REGION Network 7: Step 0 (Idle) - Warned Repark And Launch
   // Repark (0 to 30) fires only on a live occasion - the plant pre-start ParkCmd (REQ-045) or a cycle request arriving with the ram off home - and only after the pre-motion warning has sounded. Jog release deliberately triggers nothing: the ram stops and stays where it is (REQ-039, owner ruling 2026-07-16), and Off mode alone no longer self-parks an idle ram either - it parks at the next pre-start or cycle request. Launch (0 to 10) still requires the ram at home; a request with the ram off home reparks first, then launches if the request is still live at home. The two exits are mutually exclusive by construction (NOT HomeLimit vs HomeLimit, C-121).
   RUNG wire#powerrail
      Contact( #ReparkRequest )
      Contact( #JogPreStartTimer.Q )
      Move(in := 30, out1 => #IO."Step")
   END_RUNG
   RUNG wire#powerrail
      Contact( #LaunchRequest )
      Contact( #JogPreStartTimer.Q )
      Move(in := 10, out1 => #IO."Step")
   END_RUNG
   // the same network as SCL:
   IF #ReparkRequest AND #JogPreStartTimer.Q THEN #IO."Step" := 30; END_IF;
   IF #LaunchRequest AND #JogPreStartTimer.Q THEN #IO."Step" := 10; END_IF;
END_REGION

REGION Network 8: Step 10 (Drive To End Travel) - Timer, Timeout Fault, And Transitions
   // Every abnormal exit - CycleAbort (Off commanded mid-stroke, or the plant acquired a stop reason), or a timeout, whether or not it also trips Blocked - goes straight to Retract (30), never a bare stop; the ram is never left sitting mid-travel. Only reaching FullTravelLimit cleanly goes to Hold (20) first, per the normal cycle. Fitted gates the supervision timer (a disabled pusher looks for no switch feedback, REQ-043) and the fault latch (raises nothing, REQ-044).
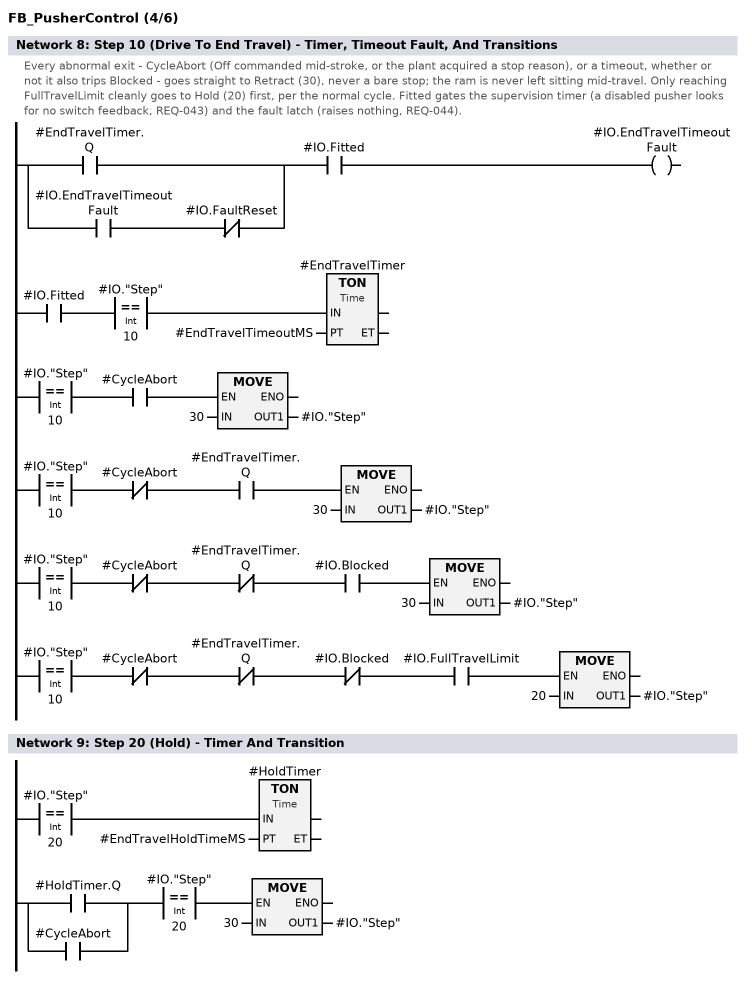
   RUNG wire#powerrail
      Contact( #EndTravelTimer.Q )
      wire#w1
      Contact( #IO.Fitted )
      Coil( #IO.EndTravelTimeoutFault )
   END_RUNG
   RUNG wire#powerrail
      Contact( #IO.EndTravelTimeoutFault )
      I_Contact( #IO.FaultReset )
   END_RUNG wire#w1
   RUNG wire#powerrail
      Contact( #IO.Fitted )
      { S7_Templates := "SrcType := Int" } EQ_Contact(in1 := #IO."Step", in2 := 10)
      { S7_Templates := "time_type := Time" } #EndTravelTimer.TON(pt := #EndTravelTimeoutMS, et =>)
   END_RUNG
   RUNG wire#powerrail
      { S7_Templates := "SrcType := Int" } EQ_Contact(in1 := #IO."Step", in2 := 10)
      Contact( #CycleAbort )
      Move(in := 30, out1 => #IO."Step")
   END_RUNG
   RUNG wire#powerrail
      { S7_Templates := "SrcType := Int" } EQ_Contact(in1 := #IO."Step", in2 := 10)
      I_Contact( #CycleAbort )
      Contact( #EndTravelTimer.Q )
      Move(in := 30, out1 => #IO."Step")
   END_RUNG
   RUNG wire#powerrail
      { S7_Templates := "SrcType := Int" } EQ_Contact(in1 := #IO."Step", in2 := 10)
      I_Contact( #CycleAbort )
      I_Contact( #EndTravelTimer.Q )
      Contact( #IO.Blocked )
      Move(in := 30, out1 => #IO."Step")
   END_RUNG
   RUNG wire#powerrail
      { S7_Templates := "SrcType := Int" } EQ_Contact(in1 := #IO."Step", in2 := 10)
      I_Contact( #CycleAbort )
      I_Contact( #EndTravelTimer.Q )
      I_Contact( #IO.Blocked )
      Contact( #IO.FullTravelLimit )
      Move(in := 20, out1 => #IO."Step")
   END_RUNG
   // the same network as SCL:
   #IO.EndTravelTimeoutFault := (#EndTravelTimer.Q OR (#IO.EndTravelTimeoutFault AND NOT #IO.FaultReset)) AND #IO.Fitted;
   #EndTravelTimer(IN := #IO.Fitted AND (#IO."Step" = 10), PT := #EndTravelTimeoutMS);   // TON
   IF (#IO."Step" = 10) AND #CycleAbort THEN #IO."Step" := 30; END_IF;
   IF (#IO."Step" = 10) AND NOT #CycleAbort AND #EndTravelTimer.Q THEN #IO."Step" := 30; END_IF;
   IF (#IO."Step" = 10) AND NOT #CycleAbort AND NOT #EndTravelTimer.Q AND #IO.Blocked THEN
       #IO."Step" := 30;
   END_IF;
   IF (#IO."Step" = 10) AND NOT #CycleAbort AND NOT #EndTravelTimer.Q AND NOT #IO.Blocked AND #IO.FullTravelLimit THEN
       #IO."Step" := 20;
   END_IF;
END_REGION

REGION Network 9: Step 20 (Hold) - Timer And Transition
   RUNG wire#powerrail
      { S7_Templates := "SrcType := Int" } EQ_Contact(in1 := #IO."Step", in2 := 20)
      { S7_Templates := "time_type := Time" } #HoldTimer.TON(pt := #EndTravelHoldTimeMS, et =>)
   END_RUNG
   RUNG wire#powerrail
      Contact( #HoldTimer.Q )
      wire#w1
      { S7_Templates := "SrcType := Int" } EQ_Contact(in1 := #IO."Step", in2 := 20)
      Move(in := 30, out1 => #IO."Step")
   END_RUNG
   RUNG wire#powerrail
      Contact( #CycleAbort )
   END_RUNG wire#w1
   // the same network as SCL:
   #HoldTimer(IN := #IO."Step" = 20, PT := #EndTravelHoldTimeMS);   // TON
   IF (#HoldTimer.Q OR #CycleAbort) AND (#IO."Step" = 20) THEN #IO."Step" := 30; END_IF;
END_REGION

REGION Network 10: Step 30 (Retract) - Timer, Timeout Fault, And Transitions
   // ParkedTimer's own Q feeds the fault latch; genuinely stuck retracting has no safer intermediate step to abort into (unlike Step 10), so the recovery transition is FaultReset AND ParkedTimeoutFault straight to Step 0 (idle) - C-123's universal FaultReset-recovery rule: a fault is never left with no transition, even when 'back to idle' is the only option. Fitted gates the supervision timer and the fault latch (REQ-043/044) - a disabled pusher neither watches for the home switch nor raises the fault.
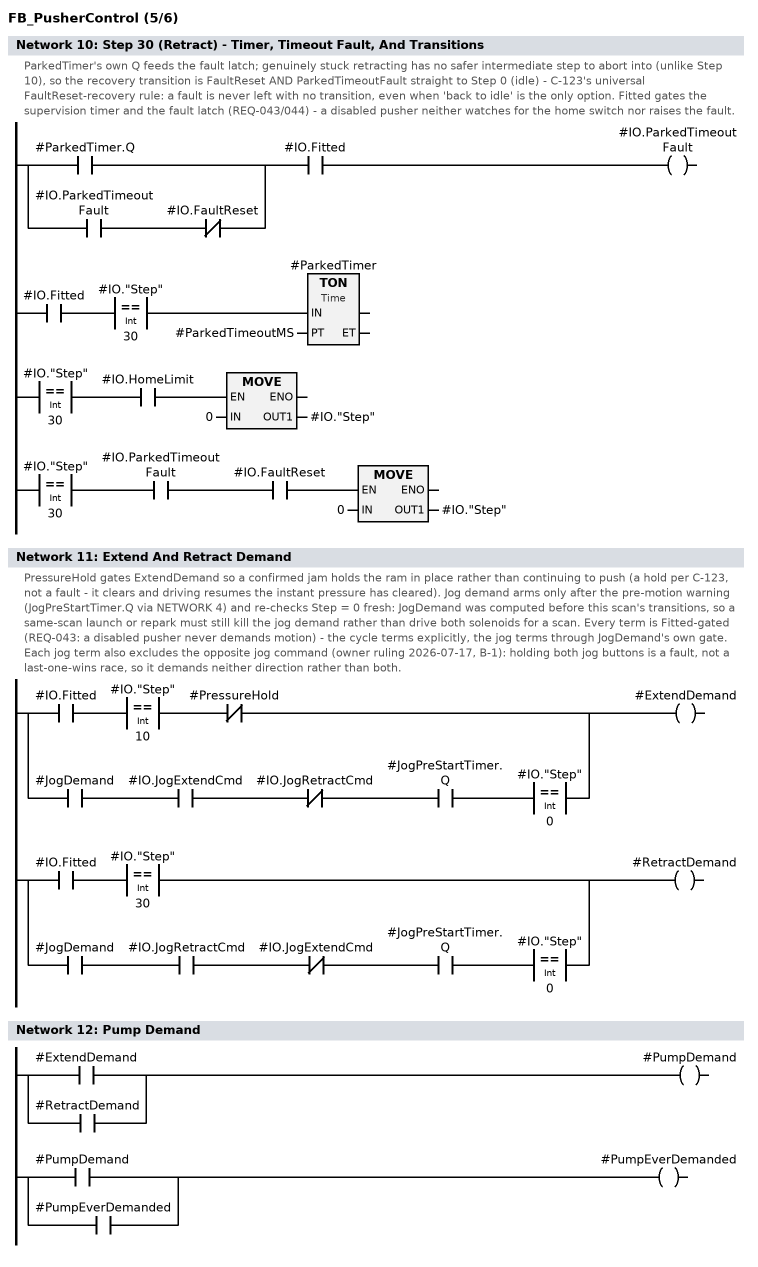
   RUNG wire#powerrail
      Contact( #ParkedTimer.Q )
      wire#w1
      Contact( #IO.Fitted )
      Coil( #IO.ParkedTimeoutFault )
   END_RUNG
   RUNG wire#powerrail
      Contact( #IO.ParkedTimeoutFault )
      I_Contact( #IO.FaultReset )
   END_RUNG wire#w1
   RUNG wire#powerrail
      Contact( #IO.Fitted )
      { S7_Templates := "SrcType := Int" } EQ_Contact(in1 := #IO."Step", in2 := 30)
      { S7_Templates := "time_type := Time" } #ParkedTimer.TON(pt := #ParkedTimeoutMS, et =>)
   END_RUNG
   RUNG wire#powerrail
      { S7_Templates := "SrcType := Int" } EQ_Contact(in1 := #IO."Step", in2 := 30)
      Contact( #IO.HomeLimit )
      Move(in := 0, out1 => #IO."Step")
   END_RUNG
   RUNG wire#powerrail
      { S7_Templates := "SrcType := Int" } EQ_Contact(in1 := #IO."Step", in2 := 30)
      Contact( #IO.ParkedTimeoutFault )
      Contact( #IO.FaultReset )
      Move(in := 0, out1 => #IO."Step")
   END_RUNG
   // the same network as SCL:
   #IO.ParkedTimeoutFault := (#ParkedTimer.Q OR (#IO.ParkedTimeoutFault AND NOT #IO.FaultReset)) AND #IO.Fitted;
   #ParkedTimer(IN := #IO.Fitted AND (#IO."Step" = 30), PT := #ParkedTimeoutMS);   // TON
   IF (#IO."Step" = 30) AND #IO.HomeLimit THEN #IO."Step" := 0; END_IF;
   IF (#IO."Step" = 30) AND #IO.ParkedTimeoutFault AND #IO.FaultReset THEN #IO."Step" := 0; END_IF;
END_REGION

REGION Network 11: Extend And Retract Demand
   // PressureHold gates ExtendDemand so a confirmed jam holds the ram in place rather than continuing to push (a hold per C-123, not a fault - it clears and driving resumes the instant pressure has cleared). Jog demand arms only after the pre-motion warning (JogPreStartTimer.Q via NETWORK 4) and re-checks Step = 0 fresh: JogDemand was computed before this scan's transitions, so a same-scan launch or repark must still kill the jog demand rather than drive both solenoids for a scan. Every term is Fitted-gated (REQ-043: a disabled pusher never demands motion) - the cycle terms explicitly, the jog terms through JogDemand's own gate. Each jog term also excludes the opposite jog command (owner ruling 2026-07-17, B-1): holding both jog buttons is a fault, not a last-one-wins race, so it demands neither direction rather than both.
   RUNG wire#powerrail
      Contact( #IO.Fitted )
      { S7_Templates := "SrcType := Int" } EQ_Contact(in1 := #IO."Step", in2 := 10)
      I_Contact( #PressureHold )
      wire#w1
      Coil( #ExtendDemand )
   END_RUNG
   RUNG wire#powerrail
      Contact( #JogDemand )
      Contact( #IO.JogExtendCmd )
      I_Contact( #IO.JogRetractCmd )
      Contact( #JogPreStartTimer.Q )
      { S7_Templates := "SrcType := Int" } EQ_Contact(in1 := #IO."Step", in2 := 0)
   END_RUNG wire#w1
   RUNG wire#powerrail
      Contact( #IO.Fitted )
      { S7_Templates := "SrcType := Int" } EQ_Contact(in1 := #IO."Step", in2 := 30)
      wire#w2
      Coil( #RetractDemand )
   END_RUNG
   RUNG wire#powerrail
      Contact( #JogDemand )
      Contact( #IO.JogRetractCmd )
      I_Contact( #IO.JogExtendCmd )
      Contact( #JogPreStartTimer.Q )
      { S7_Templates := "SrcType := Int" } EQ_Contact(in1 := #IO."Step", in2 := 0)
   END_RUNG wire#w2
   // the same network as SCL:
   #ExtendDemand := (#IO.Fitted AND (#IO."Step" = 10) AND NOT #PressureHold) OR (#JogDemand AND #IO.JogExtendCmd AND NOT #IO.JogRetractCmd AND #JogPreStartTimer.Q AND (#IO."Step" = 0));
   #RetractDemand := (#IO.Fitted AND (#IO."Step" = 30)) OR (#JogDemand AND #IO.JogRetractCmd AND NOT #IO.JogExtendCmd AND #JogPreStartTimer.Q AND (#IO."Step" = 0));
END_REGION

REGION Network 12: Pump Demand
   RUNG wire#powerrail
      Contact( #ExtendDemand )
      wire#w1
      Coil( #PumpDemand )
   END_RUNG
   RUNG wire#powerrail
      Contact( #RetractDemand )
   END_RUNG wire#w1
   RUNG wire#powerrail
      Contact( #PumpDemand )
      wire#w2
      Coil( #PumpEverDemanded )
   END_RUNG
   RUNG wire#powerrail
      Contact( #PumpEverDemanded )
   END_RUNG wire#w2
   // the same network as SCL:
   #PumpDemand := #ExtendDemand OR #RetractDemand;
   #PumpEverDemanded := #PumpDemand OR #PumpEverDemanded;
END_REGION

REGION Network 13: Pump Run-On Timer And Output Commands
   // Off-delay built from TON+inversion, not TOF/TONR (C-406). PumpEverDemanded guards a cold-start gap: on power-up PumpDemand and the timer's Q are both initially false, which would read as 'run-on already elapsed' and skip straight to no-run. RunPowerPack stays on through the run-on tail even after demand drops, but the Extend/Retract solenoids are not - they only ever follow live demand, gated by PowerPackRunningFB so the ram can't be commanded before the pump has confirmed running. Fitted gates RunPowerPack directly too: disabling the pusher must kill the pack immediately, run-on tail included (REQ-043).
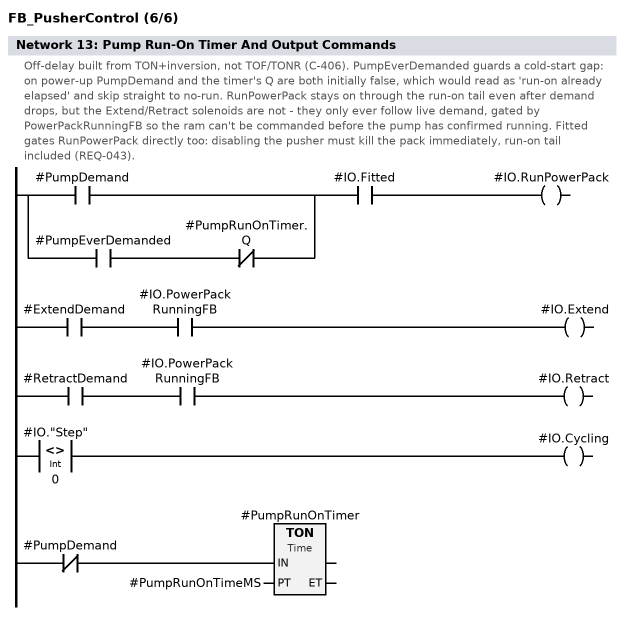
   RUNG wire#powerrail
      Contact( #PumpDemand )
      wire#w1
      Contact( #IO.Fitted )
      Coil( #IO.RunPowerPack )
   END_RUNG
   RUNG wire#powerrail
      Contact( #PumpEverDemanded )
      I_Contact( #PumpRunOnTimer.Q )
   END_RUNG wire#w1
   RUNG wire#powerrail
      Contact( #ExtendDemand )
      Contact( #IO.PowerPackRunningFB )
      Coil( #IO.Extend )
   END_RUNG
   RUNG wire#powerrail
      Contact( #RetractDemand )
      Contact( #IO.PowerPackRunningFB )
      Coil( #IO.Retract )
   END_RUNG
   RUNG wire#powerrail
      { S7_Templates := "SrcType := Int" } NE_Contact(in1 := #IO."Step", in2 := 0)
      Coil( #IO.Cycling )
   END_RUNG
   RUNG wire#powerrail
      I_Contact( #PumpDemand )
      { S7_Templates := "time_type := Time" } #PumpRunOnTimer.TON(pt := #PumpRunOnTimeMS, et =>)
   END_RUNG
   // the same network as SCL:
   #IO.RunPowerPack := (#PumpDemand OR (#PumpEverDemanded AND NOT #PumpRunOnTimer.Q)) AND #IO.Fitted;
   #IO.Extend := #ExtendDemand AND #IO.PowerPackRunningFB;
   #IO.Retract := #RetractDemand AND #IO.PowerPackRunningFB;
   #IO.Cycling := #IO."Step" <> 0;
   #PumpRunOnTimer(IN := NOT #PumpDemand, PT := #PumpRunOnTimeMS);   // TON
END_REGION
END_FUNCTION_BLOCK

FUNCTION "FC_AlarmsMain" : Void   // FC4, LAD
TITLE = Alarms Main
{ S7_Optimized_Access := 'TRUE' }
VERSION : 0.1
// stored: AutoNumber true, IsIECCheckEnabled false, SetENOAutomatically false, UDAEnableTagReadback false
BEGIN

REGION Network 1: Shredder Motor - Fault/Overload Tripped - Check Soft Starter
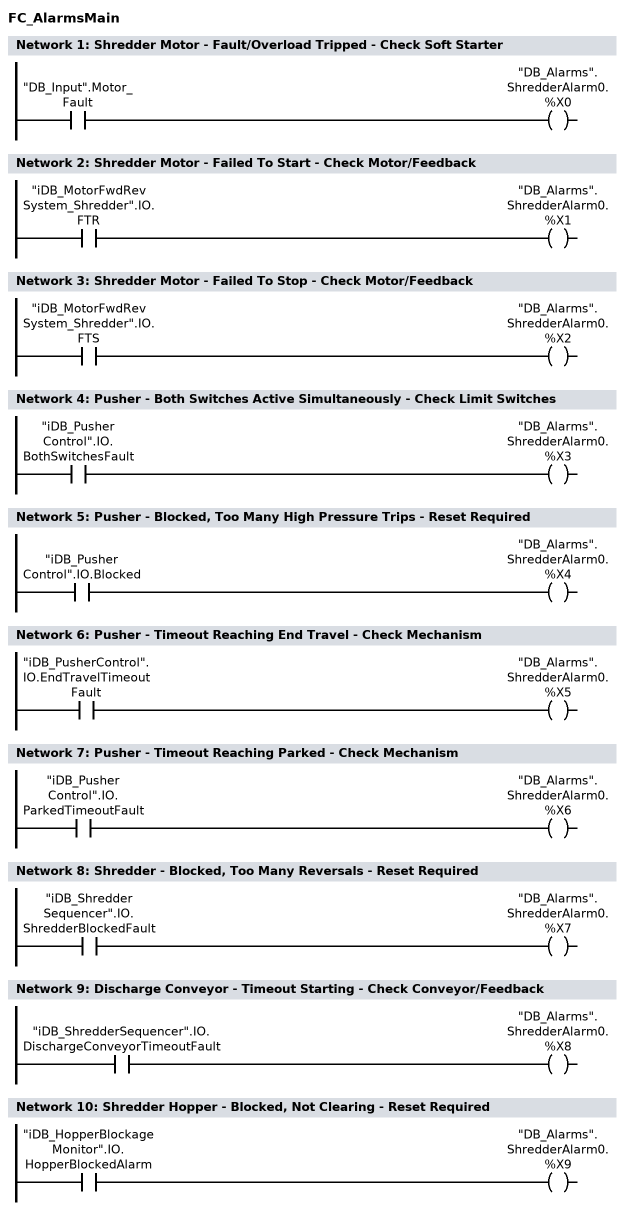
   RUNG wire#powerrail
      Contact( "DB_Input".Motor_Fault )
      Coil( "DB_Alarms".ShredderAlarm0.%X0 )
   END_RUNG
   // the same network as SCL:
   "DB_Alarms".ShredderAlarm0.%X0 := "DB_Input".Motor_Fault;
END_REGION

REGION Network 2: Shredder Motor - Failed To Start - Check Motor/Feedback
   RUNG wire#powerrail
      Contact( "iDB_MotorFwdRevSystem_Shredder".IO.FTR )
      Coil( "DB_Alarms".ShredderAlarm0.%X1 )
   END_RUNG
   // the same network as SCL:
   "DB_Alarms".ShredderAlarm0.%X1 := "iDB_MotorFwdRevSystem_Shredder".IO.FTR;
END_REGION

REGION Network 3: Shredder Motor - Failed To Stop - Check Motor/Feedback
   RUNG wire#powerrail
      Contact( "iDB_MotorFwdRevSystem_Shredder".IO.FTS )
      Coil( "DB_Alarms".ShredderAlarm0.%X2 )
   END_RUNG
   // the same network as SCL:
   "DB_Alarms".ShredderAlarm0.%X2 := "iDB_MotorFwdRevSystem_Shredder".IO.FTS;
END_REGION

REGION Network 4: Pusher - Both Switches Active Simultaneously - Check Limit Switches
   RUNG wire#powerrail
      Contact( "iDB_PusherControl".IO.BothSwitchesFault )
      Coil( "DB_Alarms".ShredderAlarm0.%X3 )
   END_RUNG
   // the same network as SCL:
   "DB_Alarms".ShredderAlarm0.%X3 := "iDB_PusherControl".IO.BothSwitchesFault;
END_REGION

REGION Network 5: Pusher - Blocked, Too Many High Pressure Trips - Reset Required
   RUNG wire#powerrail
      Contact( "iDB_PusherControl".IO.Blocked )
      Coil( "DB_Alarms".ShredderAlarm0.%X4 )
   END_RUNG
   // the same network as SCL:
   "DB_Alarms".ShredderAlarm0.%X4 := "iDB_PusherControl".IO.Blocked;
END_REGION

REGION Network 6: Pusher - Timeout Reaching End Travel - Check Mechanism
   RUNG wire#powerrail
      Contact( "iDB_PusherControl".IO.EndTravelTimeoutFault )
      Coil( "DB_Alarms".ShredderAlarm0.%X5 )
   END_RUNG
   // the same network as SCL:
   "DB_Alarms".ShredderAlarm0.%X5 := "iDB_PusherControl".IO.EndTravelTimeoutFault;
END_REGION

REGION Network 7: Pusher - Timeout Reaching Parked - Check Mechanism
   RUNG wire#powerrail
      Contact( "iDB_PusherControl".IO.ParkedTimeoutFault )
      Coil( "DB_Alarms".ShredderAlarm0.%X6 )
   END_RUNG
   // the same network as SCL:
   "DB_Alarms".ShredderAlarm0.%X6 := "iDB_PusherControl".IO.ParkedTimeoutFault;
END_REGION

REGION Network 8: Shredder - Blocked, Too Many Reversals - Reset Required
   RUNG wire#powerrail
      Contact( "iDB_ShredderSequencer".IO.ShredderBlockedFault )
      Coil( "DB_Alarms".ShredderAlarm0.%X7 )
   END_RUNG
   // the same network as SCL:
   "DB_Alarms".ShredderAlarm0.%X7 := "iDB_ShredderSequencer".IO.ShredderBlockedFault;
END_REGION

REGION Network 9: Discharge Conveyor - Timeout Starting - Check Conveyor/Feedback
   RUNG wire#powerrail
      Contact( "iDB_ShredderSequencer".IO.DischargeConveyorTimeoutFault )
      Coil( "DB_Alarms".ShredderAlarm0.%X8 )
   END_RUNG
   // the same network as SCL:
   "DB_Alarms".ShredderAlarm0.%X8 := "iDB_ShredderSequencer".IO.DischargeConveyorTimeoutFault;
END_REGION

REGION Network 10: Shredder Hopper - Blocked, Not Clearing - Reset Required
   RUNG wire#powerrail
      Contact( "iDB_HopperBlockageMonitor".IO.HopperBlockedAlarm )
      Coil( "DB_Alarms".ShredderAlarm0.%X9 )
   END_RUNG
   // the same network as SCL:
   "DB_Alarms".ShredderAlarm0.%X9 := "iDB_HopperBlockageMonitor".IO.HopperBlockedAlarm;
END_REGION
END_FUNCTION

ORGANIZATION_BLOCK "OB100"   // OB100, LAD, Startup
TITLE = Startup Reset
{ S7_Optimized_Access := 'TRUE' }
VERSION : 0.1
// Dedicated startup-reset block (C-124/C-305/C-403), run once by the CPU on every restart (warm or cold), regardless of retentivity - non-retentivity is never relied on to clear state. Forces Step back to idle (C-118/C-119) on every stepped sequencer, clears every S/R-driven and transient-run-state bit named in the fix-wave-1 B-2 finding, and force-resets DB_PLC.Simulation (C-305). Genuine fault latches - iDB_MotorFwdRevSystem_Shredder.IO.FaultActive/FTR/FTS, iDB_PusherControl.IO.Blocked/EndTravelTimeoutFault/ParkedTimeoutFault/BothSwitchesFault, iDB_ShredderSequencer.IO.ShredderBlockedFault/DischargeConveyorTimeoutFault - are deliberately excluded per C-124's carve-out: a fault needing human acknowledgement (FaultReset) still needs it after a power cycle. Closes owner-questions B-2/D-1/Q-01 and doc 06 C-128 (no automatic restart after a stop or power event).
// stored: AutoNumber true, IsIECCheckEnabled false, SetENOAutomatically false
   VAR_INPUT
      LostRetentive : Bool;   // True if retentive data are lost
      LostRTC : Bool;   // True if date and time are lost
   END_VAR
BEGIN

REGION Network 1: Shredder sequencer - force Step idle, clear transient state (C-124)
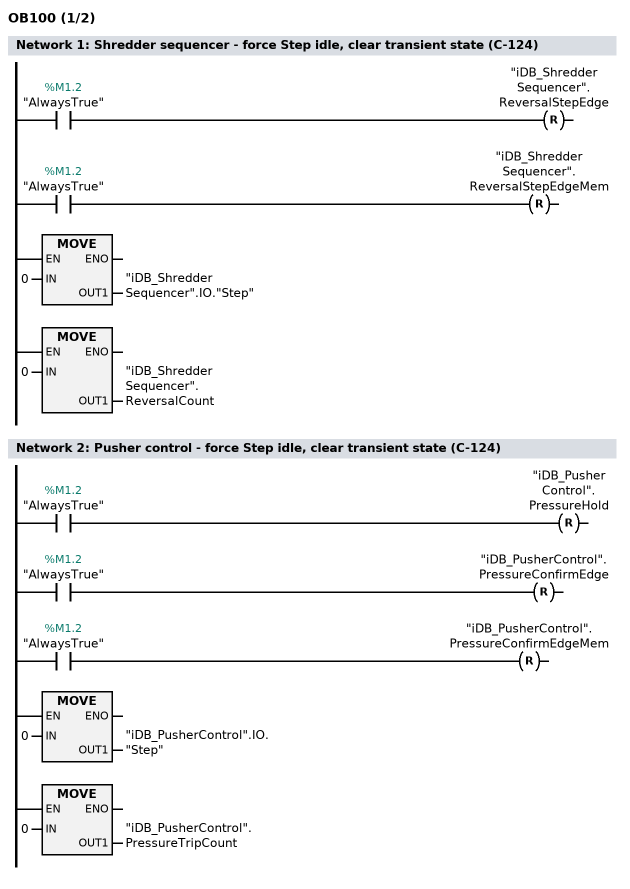
   RUNG wire#powerrail
      Contact( "AlwaysTrue" )
      R_Coil( "iDB_ShredderSequencer".ReversalStepEdge )
   END_RUNG
   RUNG wire#powerrail
      Contact( "AlwaysTrue" )
      R_Coil( "iDB_ShredderSequencer".ReversalStepEdgeMem )
   END_RUNG
   RUNG wire#powerrail
      Move(in := 0, out1 => "iDB_ShredderSequencer".IO."Step")
   END_RUNG
   RUNG wire#powerrail
      Move(in := 0, out1 => "iDB_ShredderSequencer".ReversalCount)
   END_RUNG
   // the same network as SCL:
   IF "AlwaysTrue" THEN
       "iDB_ShredderSequencer".ReversalStepEdge := FALSE;
       "iDB_ShredderSequencer".ReversalStepEdgeMem := FALSE;
   END_IF;
   "iDB_ShredderSequencer".IO."Step" := 0;
   "iDB_ShredderSequencer".ReversalCount := 0;
END_REGION

REGION Network 2: Pusher control - force Step idle, clear transient state (C-124)
   RUNG wire#powerrail
      Contact( "AlwaysTrue" )
      R_Coil( "iDB_PusherControl".PressureHold )
   END_RUNG
   RUNG wire#powerrail
      Contact( "AlwaysTrue" )
      R_Coil( "iDB_PusherControl".PressureConfirmEdge )
   END_RUNG
   RUNG wire#powerrail
      Contact( "AlwaysTrue" )
      R_Coil( "iDB_PusherControl".PressureConfirmEdgeMem )
   END_RUNG
   RUNG wire#powerrail
      Move(in := 0, out1 => "iDB_PusherControl".IO."Step")
   END_RUNG
   RUNG wire#powerrail
      Move(in := 0, out1 => "iDB_PusherControl".PressureTripCount)
   END_RUNG
   // the same network as SCL:
   IF "AlwaysTrue" THEN
       "iDB_PusherControl".PressureHold := FALSE;
       "iDB_PusherControl".PressureConfirmEdge := FALSE;
       "iDB_PusherControl".PressureConfirmEdgeMem := FALSE;
   END_IF;
   "iDB_PusherControl".IO."Step" := 0;
   "iDB_PusherControl".PressureTripCount := 0;
END_REGION

REGION Network 3: Motor FB - clear S/R-driven and transient bits (C-403), fault latches excluded
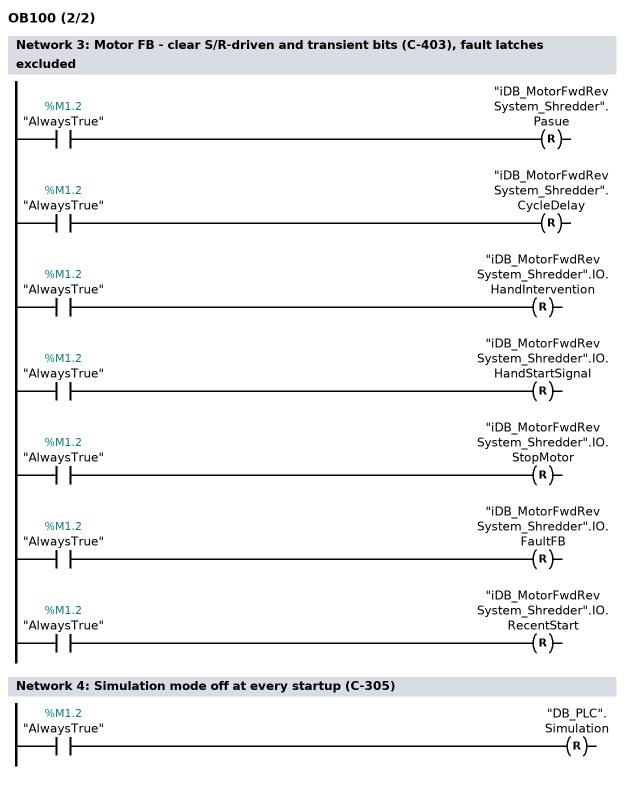
   RUNG wire#powerrail
      Contact( "AlwaysTrue" )
      R_Coil( "iDB_MotorFwdRevSystem_Shredder".Pasue )
   END_RUNG
   RUNG wire#powerrail
      Contact( "AlwaysTrue" )
      R_Coil( "iDB_MotorFwdRevSystem_Shredder".CycleDelay )
   END_RUNG
   RUNG wire#powerrail
      Contact( "AlwaysTrue" )
      R_Coil( "iDB_MotorFwdRevSystem_Shredder".IO.HandIntervention )
   END_RUNG
   RUNG wire#powerrail
      Contact( "AlwaysTrue" )
      R_Coil( "iDB_MotorFwdRevSystem_Shredder".IO.HandStartSignal )
   END_RUNG
   RUNG wire#powerrail
      Contact( "AlwaysTrue" )
      R_Coil( "iDB_MotorFwdRevSystem_Shredder".IO.StopMotor )
   END_RUNG
   RUNG wire#powerrail
      Contact( "AlwaysTrue" )
      R_Coil( "iDB_MotorFwdRevSystem_Shredder".IO.FaultFB )
   END_RUNG
   RUNG wire#powerrail
      Contact( "AlwaysTrue" )
      R_Coil( "iDB_MotorFwdRevSystem_Shredder".IO.RecentStart )
   END_RUNG
   // the same network as SCL:
   IF "AlwaysTrue" THEN
       "iDB_MotorFwdRevSystem_Shredder".Pasue := FALSE;
       "iDB_MotorFwdRevSystem_Shredder".CycleDelay := FALSE;
       "iDB_MotorFwdRevSystem_Shredder".IO.HandIntervention := FALSE;
       "iDB_MotorFwdRevSystem_Shredder".IO.HandStartSignal := FALSE;
       "iDB_MotorFwdRevSystem_Shredder".IO.StopMotor := FALSE;
       "iDB_MotorFwdRevSystem_Shredder".IO.FaultFB := FALSE;
       "iDB_MotorFwdRevSystem_Shredder".IO.RecentStart := FALSE;
   END_IF;
END_REGION

REGION Network 4: Simulation mode off at every startup (C-305)
   RUNG wire#powerrail
      Contact( "AlwaysTrue" )
      R_Coil( "DB_PLC".Simulation )
   END_RUNG
   // the same network as SCL:
   IF "AlwaysTrue" THEN "DB_PLC".Simulation := FALSE; END_IF;
END_REGION
END_ORGANIZATION_BLOCK

FUNCTION_BLOCK "FB_HopperBlockageMonitor"   // FB50, LAD
TITLE = Hopper-Blockage Monitor
{ S7_Optimized_Access := 'TRUE' }
VERSION : 0.1
// Supervises the shredder hopper high-level sensor: raises a latched hopper-blockage alarm (and a stop/inhibit demand) when the hopper stays (debounced-)high for a cumulative threshold of time while the plant is running, i.e. the shredder/pusher is not clearing it (S6 request #1, REQ-HBA-001..007). Purely supervisory - it commands no motion and writes no shared tag; the alarm and the stop demand are exposed on its own IO interface and wired to annunciation / the actual stop at a separate integration step (Q-HBA-05). Cumulative timing is pause-and-resume (NEW-HBA-01): losing PlantRunning freezes the elapsed and resumes, so 60 s of blockage need not be contiguous. Built from a plain TON, never TONR (C-406), plus a banked up-accumulator compared against the threshold (see NETWORK 3-4). The alarm latch lives in the RETAIN interface and deliberately survives a power cycle (C-124 carve-out, NEW-HBA-04) - like the sequencer's DischargeConveyorTimeoutFault, a blockage needing a human still needs FaultReset after a restart; all transient timing state is non-retentive and self-clears at startup (NEW-HBA-06, no OB100 edit). Tunables BlockedTimeThreshold (T#60S) and ClearDebounceTime (T#2S) are this instance's own settings (C-307), not shared DB members.
// stored: AutoNumber true, IsIECCheckEnabled false, IsRetainMemResEnabled false, MemoryReserve 100, SetENOAutomatically false, UDAEnableTagReadback false
   VAR RETAIN
      IO { S7_SetPoint := 'True'} : "UDT_HopperBlockageIO";   // Caller interface (C-115). Inputs (HopperLevelHigh/PlantRunning/FaultReset) are written by FC_ControlMain at integration; outputs (HopperBlockedAlarm/HopperBlockedInhibit) are read there. The whole interface is RETAIN - immaterial for the re-driven inputs, deliberate for the two output latches (C-124 carve-out).
   END_VAR
   VAR
      HighQualified : Bool;   // Debounced blockage-present latch: set the instant the hopper reads high, held through momentary sensor clears (chatter), cleared only once the hopper has read clear continuously for ClearDebounceTime (Q-HBA-02). Transient (non-retentive).
      BlockActive : Bool;   // The persistence window accrues only while this is true: a qualified blockage AND the plant actually running (Q-HBA-04).
      BlockActiveMem : Bool;   // Previous-scan BlockActive, for the constructed falling-edge (C-404).
      PauseEdge : Bool;   // One-scan pulse when BlockActive falls (plant stop or genuine clear) - fires the T_SUB bank in NETWORK 4.
      FaultResetMem : Bool;   // Previous-scan copy of the operator FaultReset input; NETWORK 5 compares the two to find the moment it goes true. Transient (non-retentive).
      FaultResetEdge : Bool;   // One-scan pulse when FaultReset goes true - the operator acknowledgement that clears the alarm latch in NETWORK 5. A reset held on produces one pulse, not a continuous clear. Transient (non-retentive).
      AccumulatedElapsed : Time;   // Cumulative high-and-running elapsed banked across plant-stop pauses (NEW-HBA-01). Two writers (NETWORK 3) that can never fire in the same scan: back to T#0S on a confirmed clear, banked up by each just-ended segment's elapsed on a plant-stop pause. A FaultReset does not touch it (REQ-HBA-005). Transient (non-retentive); starts 0, so no first-scan trip.
      CumulativeElapsed : Time;   // Live total = AccumulatedElapsed + PersistenceTimer.ET (NETWORK 4), compared against BlockedTimeThreshold to trip the alarm. Single-writer, derived each scan.
      ZeroTime : Time;   // Constant zero (T#0S) source for the accumulator reset - TIA import rejects a bare Time literal as a MOVE operand, so the zero is held as an unwritten Time member (defaults to T#0S, never written). Non-retentive.
      ClearDebounceTimer { S7_SetPoint := 'True'} : TON_TIME;
      PersistenceTimer { S7_SetPoint := 'True'} : TON_TIME;
   END_VAR
BEGIN

REGION Network 1: Confirmed-Clear Debounce
   // Times the hopper reading NOT high. Its Q (hopper clear continuously for ClearDebounceTime) is the only thing that re-arms the blockage qualifier - a shorter blip is ignored (Q-HBA-02, debounced clear).
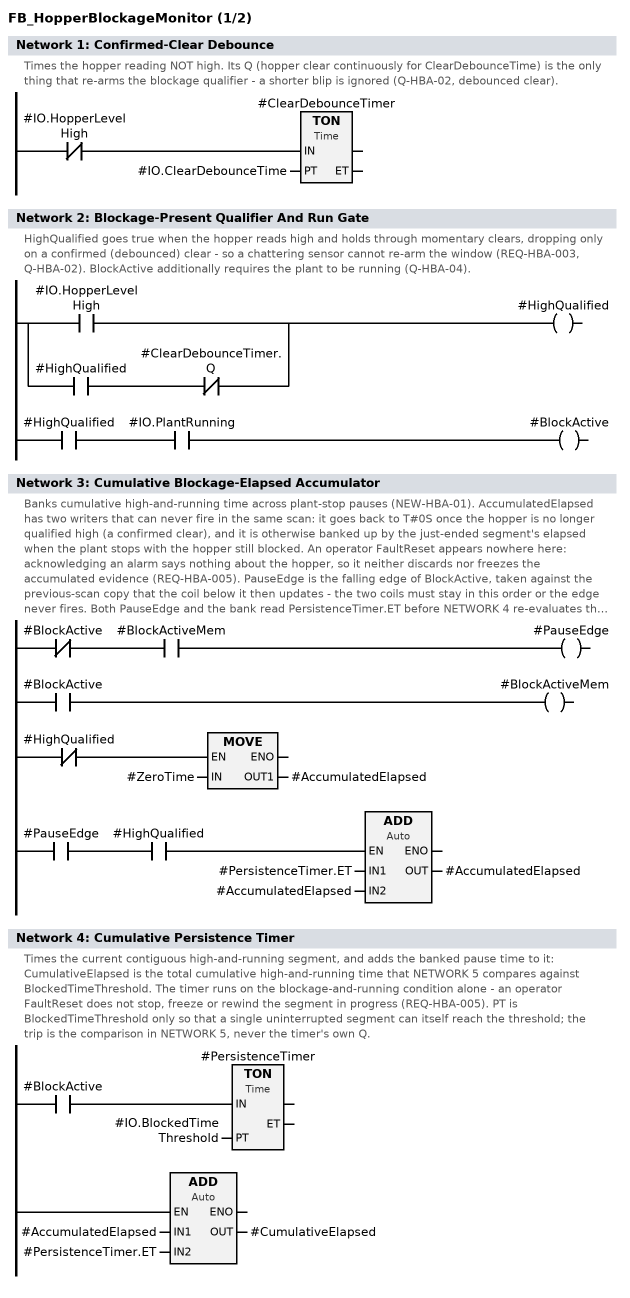
   RUNG wire#powerrail
      I_Contact( #IO.HopperLevelHigh )
      { S7_Templates := "time_type := Time" } #ClearDebounceTimer.TON(pt := #IO.ClearDebounceTime, et =>)
   END_RUNG
   // the same network as SCL:
   #ClearDebounceTimer(IN := NOT #IO.HopperLevelHigh, PT := #IO.ClearDebounceTime);   // TON
END_REGION

REGION Network 2: Blockage-Present Qualifier And Run Gate
   // HighQualified goes true when the hopper reads high and holds through momentary clears, dropping only on a confirmed (debounced) clear - so a chattering sensor cannot re-arm the window (REQ-HBA-003, Q-HBA-02). BlockActive additionally requires the plant to be running (Q-HBA-04).
   RUNG wire#powerrail
      Contact( #IO.HopperLevelHigh )
      wire#w1
      Coil( #HighQualified )
   END_RUNG
   RUNG wire#powerrail
      Contact( #HighQualified )
      I_Contact( #ClearDebounceTimer.Q )
   END_RUNG wire#w1
   RUNG wire#powerrail
      Contact( #HighQualified )
      Contact( #IO.PlantRunning )
      Coil( #BlockActive )
   END_RUNG
   // the same network as SCL:
   #HighQualified := #IO.HopperLevelHigh OR (#HighQualified AND NOT #ClearDebounceTimer.Q);
   #BlockActive := #HighQualified AND #IO.PlantRunning;
END_REGION

REGION Network 3: Cumulative Blockage-Elapsed Accumulator
   // Banks cumulative high-and-running time across plant-stop pauses (NEW-HBA-01). AccumulatedElapsed has two writers that can never fire in the same scan: it goes back to T#0S once the hopper is no longer qualified high (a confirmed clear), and it is otherwise banked up by the just-ended segment's elapsed when the plant stops with the hopper still blocked. An operator FaultReset appears nowhere here: acknowledging an alarm says nothing about the hopper, so it neither discards nor freezes the accumulated evidence (REQ-HBA-005). PauseEdge is the falling edge of BlockActive, taken against the previous-scan copy that the coil below it then updates - the two coils must stay in this order or the edge never fires. Both PauseEdge and the bank read PersistenceTimer.ET before NETWORK 4 re-evaluates the timer this scan, so the elapsed banked is the just-completed segment's, with no separate held-value register needed.
   RUNG wire#powerrail
      I_Contact( #BlockActive )
      Contact( #BlockActiveMem )
      Coil( #PauseEdge )
   END_RUNG
   RUNG wire#powerrail
      Contact( #BlockActive )
      Coil( #BlockActiveMem )
   END_RUNG
   RUNG wire#powerrail
      I_Contact( #HighQualified )
      Move(in := #ZeroTime, out1 => #AccumulatedElapsed)
   END_RUNG
   RUNG wire#powerrail
      Contact( #PauseEdge )
      Contact( #HighQualified )
      Add(in1 := #PersistenceTimer.ET, in2 := #AccumulatedElapsed, out => #AccumulatedElapsed)
   END_RUNG
   // the same network as SCL:
   #PauseEdge := NOT #BlockActive AND #BlockActiveMem;
   #BlockActiveMem := #BlockActive;
   IF NOT #HighQualified THEN #AccumulatedElapsed := #ZeroTime; END_IF;
   IF #PauseEdge AND #HighQualified THEN
       #AccumulatedElapsed := #PersistenceTimer.ET + #AccumulatedElapsed;
   END_IF;
END_REGION

REGION Network 4: Cumulative Persistence Timer
   // Times the current contiguous high-and-running segment, and adds the banked pause time to it: CumulativeElapsed is the total cumulative high-and-running time that NETWORK 5 compares against BlockedTimeThreshold. The timer runs on the blockage-and-running condition alone - an operator FaultReset does not stop, freeze or rewind the segment in progress (REQ-HBA-005). PT is BlockedTimeThreshold only so that a single uninterrupted segment can itself reach the threshold; the trip is the comparison in NETWORK 5, never the timer's own Q.
   RUNG wire#powerrail
      Contact( #BlockActive )
      { S7_Templates := "time_type := Time" } #PersistenceTimer.TON(pt := #IO.BlockedTimeThreshold, et =>)
   END_RUNG
   RUNG wire#powerrail
      Add(in1 := #AccumulatedElapsed, in2 := #PersistenceTimer.ET, out => #CumulativeElapsed)
   END_RUNG
   // the same network as SCL:
   #PersistenceTimer(IN := #BlockActive, PT := #IO.BlockedTimeThreshold);   // TON
   #CumulativeElapsed := #AccumulatedElapsed + #PersistenceTimer.ET;
END_REGION

REGION Network 5: Hopper-Blocked Alarm Latch (RETAIN - Survives Power Cycle)
   // Latches the hopper-blockage alarm when the cumulative high-and-running time reaches BlockedTimeThreshold, and holds it until an operator acknowledges. The acknowledgement is the moment FaultReset goes true, not the fact that it is true: a reset left on, wired on or stuck on clears the latch once and cannot hold the alarm off afterwards (REQ-HBA-005). Because the reset leaves the accumulated evidence alone, the latch re-evaluates on the very next scan against that same evidence - a hopper still blocked past the threshold re-alarms at once, whether or not the plant is running, while a hopper whose evidence has been discarded stays quiet. The reset pulse is taken against the previous-scan copy that the coil below it then updates - the two coils must stay in this order or the pulse never fires. The latch lives in the RETAIN interface and survives a power cycle: a blockage that needed a human still needs acknowledging after a restart, and the stop demand below stays asserted until it gets one.
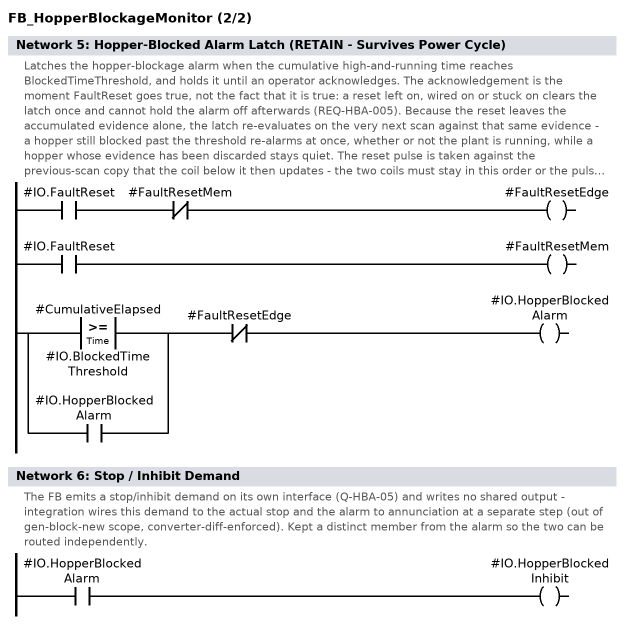
   RUNG wire#powerrail
      Contact( #IO.FaultReset )
      I_Contact( #FaultResetMem )
      Coil( #FaultResetEdge )
   END_RUNG
   RUNG wire#powerrail
      Contact( #IO.FaultReset )
      Coil( #FaultResetMem )
   END_RUNG
   RUNG wire#powerrail
      { S7_Templates := "SrcType := Time" } GE_Contact(in1 := #CumulativeElapsed, in2 := #IO.BlockedTimeThreshold)
      wire#w1
      I_Contact( #FaultResetEdge )
      Coil( #IO.HopperBlockedAlarm )
   END_RUNG
   RUNG wire#powerrail
      Contact( #IO.HopperBlockedAlarm )
   END_RUNG wire#w1
   // the same network as SCL:
   #FaultResetEdge := #IO.FaultReset AND NOT #FaultResetMem;
   #FaultResetMem := #IO.FaultReset;
   #IO.HopperBlockedAlarm := ((#CumulativeElapsed >= #IO.BlockedTimeThreshold) OR #IO.HopperBlockedAlarm) AND NOT #FaultResetEdge;
END_REGION

REGION Network 6: Stop / Inhibit Demand
   // The FB emits a stop/inhibit demand on its own interface (Q-HBA-05) and writes no shared output - integration wires this demand to the actual stop and the alarm to annunciation at a separate step (out of gen-block-new scope, converter-diff-enforced). Kept a distinct member from the alarm so the two can be routed independently.
   RUNG wire#powerrail
      Contact( #IO.HopperBlockedAlarm )
      Coil( #IO.HopperBlockedInhibit )
   END_RUNG
   // the same network as SCL:
   #IO.HopperBlockedInhibit := #IO.HopperBlockedAlarm;
END_REGION
END_FUNCTION_BLOCK

DATA_BLOCK "iDB_HopperBlockageMonitor"   // DB51
VERSION : 0.1
// Single instance of FB_HopperBlockageMonitor (S6 request #1, hopper-blockage alarm). Members mirror the FB STATIC section; BlockedTimeThreshold (T#60S) and ClearDebounceTime (T#2S) carry the commissioning defaults (C-307/C-309). Hand-authored per the compile-error-playbook's synthesize-produced-FB path.
// stored: AutoNumber true, DBAccessibleFromOPCUA true, InstanceOfName FB_HopperBlockageMonitor, InstanceOfType FB
"FB_HopperBlockageMonitor"
BEGIN
   IO.BlockedTimeThreshold := T#60S;
   IO.ClearDebounceTime := T#2S;
END_DATA_BLOCK

DATA_BLOCK "iDB_MotorFwdRevSystem_Shredder"   // DB6
VERSION : 0.1
// stored: AutoNumber true, DBAccessibleFromOPCUA true, InstanceOfName FB_MotorFwdRevSystem, InstanceOfType FB
"FB_MotorFwdRevSystem"
   // VAR RETAIN
   //    IO : "MotorFwdRevIOSet";
   // END_VAR
   // VAR
   //    RisingEdgeFlags : Array[0..3] of Bool;
   //    NegitiveSignalEdge : Array[0..2] of Bool;
   //    Pasue : Bool;
   //    HrTotaliserTimerReset : Bool;
   //    EnableUPSTimeMS : DInt;
   //    ShutdownTimeMS : DInt;
   //    FTTimeMS : DInt;
   //    PauseTimeMS : DInt;
   //    ReverseIgnoreFTTimeMS : DInt;
   //    FaultTripTimer { S7_SetPoint := 'True'} : TON_TIME;
   //    FTSTimer { S7_SetPoint := 'True'} : TON_TIME;
   //    EnableUpstreamTimer { S7_SetPoint := 'True'} : TON_TIME;
   //    ShutdownTimer { S7_SetPoint := 'True'} : TON_TIME;
   //    GeneralDelayTimer { S7_SetPoint := 'True'} : TON_TIME;
   //    InHandReqPreStart { S7_SetPoint := 'True'} : TON_TIME;
   //    CycleDelayReset { S7_SetPoint := 'True'} : TON_TIME;
   // END_VAR
   // VAR RETAIN
   //    HrTotaliserTimer { S7_SetPoint := 'True'} : TONR_TIME;
   // END_VAR
   // VAR
   //    ReversalPauseTimer { S7_SetPoint := 'True'} : TON_TIME;
   //    ReversalIgnoreFTTimer { S7_SetPoint := 'True'} : TON_TIME;
   //    PreStartMemory { S7_SetPoint := 'True'} : Bool;
   //    HandPosEdge : Bool;
   //    HandNegEdge : Bool;
   //    CycleDelay : Bool;
   // END_VAR
BEGIN
   IO.FTTime := 10.0;
   IO.ReverseDelay := 8.0;
   IO.ReverseIgnoreFT := 12.0;
END_DATA_BLOCK

DATA_BLOCK "iDB_PusherControl"   // DB10
VERSION : 0.1
// stored: AutoNumber true, DBAccessibleFromOPCUA true, InstanceOfName FB_PusherControl, InstanceOfType FB
"FB_PusherControl"
BEGIN
END_DATA_BLOCK

DATA_BLOCK "iDB_ShredderSequencer"   // DB11
VERSION : 0.1
// stored: AutoNumber true, DBAccessibleFromOPCUA true, InstanceOfName FB_ShredderSequencer, InstanceOfType FB
"FB_ShredderSequencer"
BEGIN
END_DATA_BLOCK
